TYPE ST_MainPwrPhases_HWI :
STRUCT
  L1 : ST_PhaseInfo;
  L2 : ST_PhaseInfo;
  L3 : ST_PhaseInfo;
  Tot : ST_PhasesCommon;
END_STRUCT
END_TYPE

(* stored: Version 1.1.0.1, ProductVersion 3.1.4024.12
   DUT ST_MainPwrPhases_HWI: Id {7f41b6b8-0ede-440a-b3a0-8a26c57e04c2} *)
